FUNCTION_BLOCK PUBLIC FB_Conv2
VAR_INPUT

END_VAR
VAR_OUTPUT

END_VAR
VAR
	Set_Motor	:	BOOL		;
	Reset_Motor	:	BOOL		;
	iSTEP		:	INT := 0	;
	Timer1		:	TON			;
	Timer2		:	TON			;
	Timer3		:	TON			;
	Timer4		:	TON			;
	Timer5		:	TON			;
END_VAR

CASE iSTEP OF 

	// ================================================ conv2 motor init
	0:	IF IO.bConv_Ready AND IO_control.bEstop THEN
			IO_control.bMotor2 := FALSE;
			iSTEP := iSTEP + 1;
		END_IF
	
	// ================================================ check for open status for next conv	
	1:	IF IO_Conveyor.bExit2_IsOpen THEN		
			iSTEP := iSTEP + 1;
		END_IF
	
	// ================================================ motor1 to start if conv1 job done
	2:	IF IO_Conveyor.Conv1_Done THEN
			IO_control.bMotor1 S= IO_Conveyor.Conv1_Done;
			IO_control.bMotor2 S= IO_Conveyor.Conv1_Done;
			iSTEP := iSTEP + 1;
		END_IF	
	
	// ================================================ motor1 to stop if conv2_in is ON		
	3:	IF IO.bConv2_In THEN
			IO_control.bMotor1 R= IO.bConv2_In;
			IO_Conveyor.Conv1_Done := FALSE ;
			iSTEP := iSTEP + 1 ;
		END_IF	
	
	// ================================================ stop motor if conv2_out ON	
	4:	IF IO.bConv2_Out THEN
			IO_Conveyor.Bin_At_Exit_2 := TRUE;
			IO_control.bMotor2 R= IO_Conveyor.Bin_At_Exit_2 ;
			IO_Conveyor.Conv2_Done := TRUE;
			iSTEP := iSTEP + 1 ;
		END_IF
	
	// ================================================ receive feedback from conv3	
	5:	IF NOT IO_Conveyor.Conv2_Done THEN
			iSTEP := 0 ;
		END_IF

END_CASE

IF IO_control.bReset AND IO.bManualMode THEN
	IO_Conveyor.Conv2_Done := FALSE;
	IO_Conveyor.Bin_At_Exit_2 := FALSE;
	iSTEP := 0 ;
END_IF

END_FUNCTION_BLOCK

(* stored: Version 1.1.0.1, ProductVersion 3.1.4024.12
   POU FB_Conv2: Id {78765a87-ea98-475f-b5cc-949ea656d831}, SpecialFunc None *)
